// TIA Portal V19 export
DATA_BLOCK "DB_DP_Error"   // DB203
{ S7_Optimized_Access := 'FALSE' }
// stored: AutoNumber false
   VAR
      DP_Slave : Array[0..1023] of Byte;   // 0..n.v.,nicht projektiert,1..vorhanden,ok,2..vorhanden,nok,3..projektiert,n.v.
      Altwert : Array[0..1023] of Byte;   // 0..n.v.,nicht projektiert,1..vorhanden,ok,2..vorhanden,nok,3..projektiert,n.v.
      HiAdr : Int;   // höchste Teilnehmeradresse
      Init : Bool;   // Anlaufzyklus oder AMS-Reset --> Initialisierung
      Hupe_enable : Bool;   // * Hupe bei Alarm einschalten?
      Sammelstoerung : Bool;   // Störung/Ausfall
      Sammelwarnung : Bool;   // Warnung/Fehler einer Baugruppe
      res1 : Bool;
      res2 : Bool;
      res3 : Bool;
      res4 : Bool;
   END_VAR
BEGIN
END_DATA_BLOCK
